{attribute 'linkalways'} 
{attribute 'no_explicit_call' := 'This FB is a CLASS and must be accessed using methods or properties'}
{attribute 'enable_dynamic_creation'}
FUNCTION_BLOCK _ETcVnDistanceType EXTENDS EnumDatatypeBase
VAR
	localData : ETcVnDistanceType;
	activeData : REFERENCE TO ETcVnDistanceType;
	enumBaseDatatype : _DINT(localData);
END_VAR

METHOD PRIVATE AddLocalEnumeration
VAR_INPUT
	Enumeration : T_MAXSTRING;
	Value : ETcVnDistanceType;
END_VAR
AddEnumeration(Enumeration, Value);
END_METHOD

PROPERTY PUBLIC Address : PVOID
GET
Address := ADR(activeData);
END_GET
END_PROPERTY

METHOD PUBLIC ClearReference
VAR_INPUT
END_VAR
activeData REF= localData;
SetBaseDatatypeReference();
END_METHOD

METHOD PUBLIC Clone : I_Datatype
VAR
    pClone : POINTER TO _ETcVnDistanceType;
END_VAR
pClone := __NEW(_ETcVnDistanceType(InitialValue := Value));
Clone := pClone^;
END_METHOD

METHOD FB_init : BOOL
VAR_INPUT
	bInitRetains : BOOL; // if TRUE, the retain variables are initialized (warm start / cold start)
	bInCopyCode : BOOL;  // if TRUE, the instance afterwards gets moved into the copy code (online change)
	InitialValue : ETcVnDistanceType;
END_VAR
localData := InitialValue;
AddBaseDatatype(enumBaseDatatype);
ClearReference();

AddLocalEnumeration('TCVN_DT_USER', ETcVnDistanceType.TCVN_DT_USER);
AddLocalEnumeration('TCVN_DT_L1', ETcVnDistanceType.TCVN_DT_L1);
AddLocalEnumeration('TCVN_DT_L2', ETcVnDistanceType.TCVN_DT_L2);
AddLocalEnumeration('TCVN_DT_C', ETcVnDistanceType.TCVN_DT_C);
AddLocalEnumeration('TCVN_DT_L12', ETcVnDistanceType.TCVN_DT_L12);
AddLocalEnumeration('TCVN_DT_FAIR', ETcVnDistanceType.TCVN_DT_FAIR);
AddLocalEnumeration('TCVN_DT_WELSCH', ETcVnDistanceType.TCVN_DT_WELSCH);
AddLocalEnumeration('TCVN_DT_HUBER', ETcVnDistanceType.TCVN_DT_HUBER);
END_METHOD

PROPERTY PUBLIC Identifier : T_MAXSTRING
GET
Identifier := 'ETcVnDistanceType';
END_GET
END_PROPERTY

METHOD IsEnumeratorValueEqual : BOOL
VAR_INPUT
	Enumerator : I_KeyValueForwardEnumerator;
END_VAR
VAR
	storedValue : ETcVnDistanceType;
END_VAR
IF NOT Enumerator.TryGet(storedValue) THEN
	RETURN;
END_IF

IsEnumeratorValueEqual := storedValue = activeData;
END_METHOD

METHOD PUBLIC MakeReferenceTo
VAR_INPUT
	ReferenceTarget : REFERENCE TO ETcVnDistanceType;
END_VAR
activeData REF= ReferenceTarget;
SetBaseDatatypeReference();
END_METHOD

METHOD PROTECTED SetBaseDatatypeReference
VAR_INPUT
END_VAR
enumBaseDatatype.MakeReferenceTo(activeData);
END_METHOD

PROPERTY PUBLIC Size : UDINT
GET
Size := SIZEOF(activeData);
END_GET
END_PROPERTY

METHOD TryMakeReferenceTo : BOOL
VAR_INPUT
	Target : I_Datatype;
END_VAR
VAR
	pTargetData : POINTER TO ETcVnDistanceType;
END_VAR
IF NOT IsEquivalentTo(Target) THEN
	RETURN;
END_IF

pTargetData := Target.Address;
activeData REF= pTargetData^;
SetBaseDatatypeReference();
TryMakeReferenceTo := TRUE;
END_METHOD

PROPERTY PUBLIC Value : ETcVnDistanceType
GET
Value := activeData;
END_GET
SET
activeData := Value;
END_SET
END_PROPERTY

METHOD PUBLIC TryDeserializeFrom : BOOL
VAR_INPUT
    Deserializer : I_Deserializer;
    Feedback : I_DeserializerFeedback;
END_VAR
VAR
    key : T_MAXSTRING;
END_VAR
// Accept the label emitted by older versions, but serialize the canonical label.
IF NOT Deserializer.TryGetString(key, Feedback) THEN
    RETURN;
END_IF

IF key = 'TCVN_DT_HUBER ' THEN
    activeData := ETcVnDistanceType.TCVN_DT_HUBER;
    TryDeserializeFrom := TRUE;
    RETURN;
END_IF

TryDeserializeFrom := SUPER^.TryDeserializeFrom(Deserializer, Feedback);
END_METHOD

END_FUNCTION_BLOCK

(* stored: Version 1.1.0.1, ProductVersion 3.1.4024.13
   POU _ETcVnDistanceType: Id {2e4ff358-7934-033a-1437-30de61b51c55}, SpecialFunc None
   Folder Core: Id {ddfd9a77-2220-0ce2-381e-93f0d9f98edb}
   Folder Protected: Id {4919a46e-ec2e-017d-2cde-a23e7b9ca592}
   Folder Customize: Id {dc195db8-5342-0e30-13d6-1cee201c21f4}
   Folder Constructor: Id {405fbe48-eaaa-0b80-1a38-433bbbfa0c52}
   Folder Private: Id {f8f01058-915c-04ff-2bec-d8f9f2847444}
   Folder Protected: Id {a10a2415-6be2-0048-3606-47191fefcfe6}
   Method AddLocalEnumeration: Id {89227239-77c5-0940-03f5-fedeb7649da7}
   Property Address: Id {a87564b7-2d9e-02df-3295-e82cfdfd3f8d}
   Get Get: Id {5ddcd883-1073-0459-0639-f4c8d5f73921}
   Method ClearReference: Id {77505507-1e08-0dca-018e-6e1bb33912ec}
   Method Clone: Id {21f09ad7-97e0-08a3-39aa-17f097455468}
   Method FB_init: Id {555cd26e-0b45-00ee-0938-5d14bc15af77}
   Property Identifier: Id {c0c0b2f9-e0c3-07d1-39b7-943db26a0193}
   Get Get: Id {f9544924-0886-0499-3d05-475e63e9db68}
   Method IsEnumeratorValueEqual: Id {c74fb5eb-5d6d-0b78-1134-99ad7e435d97}
   Method MakeReferenceTo: Id {a9f7882c-a738-01b0-33bd-d59082fae296}
   Method SetBaseDatatypeReference: Id {53e28781-83f6-0940-2b96-4612279b3840}
   Property Size: Id {6640ec96-5906-0a1e-2c3b-d24e2a82403a}
   Get Get: Id {2528d1bb-1f2a-09df-2bf9-e0a041a5a95c}
   Method TryMakeReferenceTo: Id {fe86513d-1037-052d-3e0c-27e711c504b8}
   Property Value: Id {7c66437f-87e3-0279-3505-cda71ecea50d}
   Get Get: Id {2ce33f8b-ac38-0c64-2576-95c3b9f170d3}
   Set Set: Id {81d4ec10-a201-0beb-16f5-b959f888e93b}
   Method TryDeserializeFrom: Id {34d65c73-1b93-470b-a73a-a0765a6a28e6} *)
